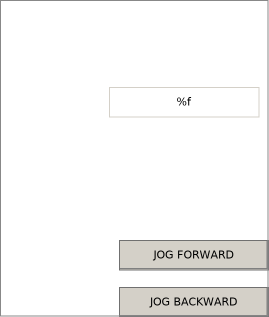
VISUALIZATION Visualization  // 269x317
    Button (119,287 150x30), "JOG BACKWARD"
        tap GVL.bJogBackward
    Button (119,240 150x30), "JOG FORWARD"
        tap GVL.bJogForward
    Textfield (109,87 150x30), "%f", text variable: MAIN.AxisControlConv1.fbMCReadActPos.Position
END_VISUALIZATION

(* stored: Version 1.1.0.1, ProductVersion 3.1.4024.15
   Visu Visualization: Id {69e0c124-467e-426d-8304-62869b83219a} *)
